PROGRAM MAIN
VAR
END_VAR

PRG_ALARMS();	//Chamada do programa Alarmes / call program ALARMS

END_PROGRAM

(* stored: Version 1.1.0.1, ProductVersion 3.1.4024.12
   POU MAIN: Id {0a7fe922-6658-48a1-87b6-5b2f1ace9db1}, SpecialFunc None *)
